// TIA Portal V19 export
DATA_BLOCK "DEBUG"   // DB124
// stored: Access Published, MemoryReserve 100
   VAR
      Force_Sinamics_Infeed_ON : Bool;
      Alr { S7_SetPoint := 'True'} : Array[1..10] of Bool;
      Core_iSlaveSynchPos : LReal;
      "Core.iMasterSyncPos" : LReal;
      "Core.iWorkPosition" : LReal;
      "Core.SlavePosition" : LReal;
   END_VAR
BEGIN
END_DATA_BLOCK
